{attribute 'linkalways'} 
{attribute 'no_explicit_call' := 'This FB is a CLASS and must be accessed using methods or properties'}
{attribute 'enable_dynamic_creation'}
FUNCTION_BLOCK INTERNAL AsyncCommandStateMachine IMPLEMENTS I_AsyncCommandStateControl
VAR
	state : (IDLE, INITIALIZING, EXECUTING, COMPLETING, COMPLETED, ABORTING, ABORTED, ERRORED);
	_errorId : UDINT;
END_VAR

(*
State Machine
    ┌──────┐
    │ Idle │
    └──┬───┘
       │                    Error
       │ Execute           ┌────────────────────────────────────────┐
       │                   │                                        │
┌──────▼───────┐ Next ┌────┴──────┐ Next ┌────────────┐ Error       │
│ Initializing ├──────► Executing ├──────► Completing ├──────────┐  │
└──────┬───────┘      └────┬──────┘      └─────┬──────┘          │  │
       │                   │                   │                 │  │
       │ Error             │ Abort             │ Next            │  │
       │                   │                   │                 │  │
       │              ┌────▼─────┐ Error       │                 │  │
       │              │ Aborting ├─────────────┼──────────────┐  │  │
       │              └────┬─────┘             │              │  │  │
       │                   │                   │              │  │  │
       │                   │ Next              │              │  │  │
       │                   │                   │              │  │  │
       │              ┌────▼────┐        ┌─────▼─────┐      ┌─▼──▼──▼─┐
       │              │ Aborted │        │ Completed │      │ Errored │
       │              └─────────┘        └───────────┘      └────▲────┘
       │                                                         │
       └─────────────────────────────────────────────────────────┘
*)

METHOD PUBLIC Abort
CASE state OF
	IDLE : RETURN;
	ABORTING : RETURN;
	COMPLETED : RETURN;
	ABORTED : RETURN;
	ERRORED : RETURN;
END_CASE

state := ABORTING;
END_METHOD

METHOD PUBLIC Error
VAR_INPUT
	errorId : UDINT;
END_VAR
CASE state OF
	IDLE : RETURN;
	COMPLETED : RETURN;
	ABORTED : RETURN;
	ERRORED : RETURN;
END_CASE

_errorId := errorId;
state := ERRORED;
END_METHOD

{attribute 'monitoring' := 'call'}
PROPERTY PUBLIC ErrorId : UDINT
GET // PUBLIC
ErrorId := _errorId;
END_GET
END_PROPERTY

METHOD PUBLIC Execute
CASE state OF
	INITIALIZING : RETURN;
	EXECUTING : RETURN;
	COMPLETING : RETURN;
	ABORTING : RETURN;
END_CASE

_errorId := 0;
state := INITIALIZING;
END_METHOD

{attribute 'monitoring' := 'call'}
PROPERTY PUBLIC IsAborted : BOOL
GET // PUBLIC
IsAborted := state = ABORTED;
END_GET
END_PROPERTY

{attribute 'monitoring' := 'call'}
PROPERTY PUBLIC IsAborting : BOOL
GET // PUBLIC
IsAborting := state = ABORTING;
END_GET
END_PROPERTY

{attribute 'monitoring' := 'call'}
PROPERTY PUBLIC IsCompleted : BOOL
GET // PUBLIC
IsCompleted := state = COMPLETED;
END_GET
END_PROPERTY

{attribute 'monitoring' := 'call'}
PROPERTY PUBLIC IsCompleting : BOOL
GET // PUBLIC
IsCompleting := state = COMPLETING;
END_GET
END_PROPERTY

{attribute 'monitoring' := 'call'}
PROPERTY PUBLIC IsErrored : BOOL
GET // PUBLIC
IsErrored := state = ERRORED;
END_GET
END_PROPERTY

{attribute 'monitoring' := 'call'}
PROPERTY PUBLIC IsExecuting : BOOL
GET // PUBLIC
IsExecuting := state = EXECUTING;
END_GET
END_PROPERTY

{attribute 'monitoring' := 'call'}
PROPERTY PUBLIC IsIdle : BOOL
GET // PUBLIC
IsIdle:= state = IDLE;
END_GET
END_PROPERTY

{attribute 'monitoring' := 'call'}
PROPERTY PUBLIC IsInitializing : BOOL
GET // PUBLIC
IsInitializing := state = INITIALIZING;
END_GET
END_PROPERTY

METHOD PUBLIC Next
CASE state OF
	IDLE : RETURN;
	INITIALIZING : StateComplete_Initializing();
	EXECUTING : StateComplete_Executing();
	COMPLETING : StateComplete_Completing();
	COMPLETED : RETURN;
	ABORTING : StateComplete_Aborting();
	ABORTED : RETURN;
	ERRORED : RETURN;
END_CASE
END_METHOD

METHOD PRIVATE StateComplete_Aborting
state := ABORTED;
END_METHOD

METHOD PRIVATE StateComplete_Completing
state := COMPLETED;
END_METHOD

METHOD PRIVATE StateComplete_Executing
state := COMPLETING;
END_METHOD

METHOD PRIVATE StateComplete_Initializing
state := EXECUTING;
END_METHOD

END_FUNCTION_BLOCK

(* stored: Version 1.1.0.1, ProductVersion 3.1.4024.12
   POU AsyncCommandStateMachine: Id {d31cc0cc-16b4-4b07-a6af-35ddcb7c0711}, SpecialFunc None
   Folder Private: Id {41426bd1-a226-0803-0384-e062ce7381b2}
   Method Abort: Id {78c22115-5b85-0d50-1bd1-09ca78ea3fd1}
   Method Error: Id {18d6a5d8-96f4-0214-2b15-d10a997ecb87}
   Property ErrorId: Id {c5ec3162-ba6d-041d-3f3c-c8f5993b84e7}
   Get Get: Id {c877bd70-7bda-0b3e-2ccc-7a7e50987718}
   Method Execute: Id {bc66cba2-0366-0798-2fcd-65188d719db8}
   Property IsAborted: Id {9935f71d-980f-0975-0522-8cc4cbfb75ea}
   Get Get: Id {0b2a1cf9-e737-0465-344d-50e5bbae51d3}
   Property IsAborting: Id {04b092b0-40e8-054e-1f50-cd6f844876e9}
   Get Get: Id {905ff163-f255-0bb7-1496-a0c9db2fa59a}
   Property IsCompleted: Id {62fa8999-a6c2-09ff-3455-85d275619a26}
   Get Get: Id {050dcc6f-5274-0b30-048a-94757015eedd}
   Property IsCompleting: Id {ff6612e9-4498-0e9a-1cf5-4b43e2da028d}
   Get Get: Id {759252e6-f179-0cda-3559-75be88189814}
   Property IsErrored: Id {ff93ab43-ebf2-0230-3d19-f222afd8bcc2}
   Get Get: Id {6bee74d6-703e-042a-1fca-320563290093}
   Property IsExecuting: Id {36c34b42-44ed-01ea-1888-6178766ddcd4}
   Get Get: Id {ef95ac24-4c50-0c56-2905-a8c914749852}
   Property IsIdle: Id {52586fe8-a9c9-0414-265f-2080ea24f1de}
   Get Get: Id {8c14f0a1-91b4-00bf-2d9c-4577b31a3c5b}
   Property IsInitializing: Id {99dd60cc-4abe-0fbc-1f74-698bcb0f7322}
   Get Get: Id {c1662816-4e65-022c-0b2a-e6d27dfe215c}
   Method Next: Id {d4c73f06-c16b-00f1-1b40-d28d4a8d0e71}
   Method StateComplete_Aborting: Id {5258c404-ec4e-0960-077c-91eb2bfaf45c}
   Method StateComplete_Completing: Id {46e85e9c-fd98-0aa7-32ec-c6a472347e8d}
   Method StateComplete_Executing: Id {11c2ac65-de78-0d43-185f-d15738abfb29}
   Method StateComplete_Initializing: Id {9112795b-6bf9-0d9e-0480-40f30f283991} *)
